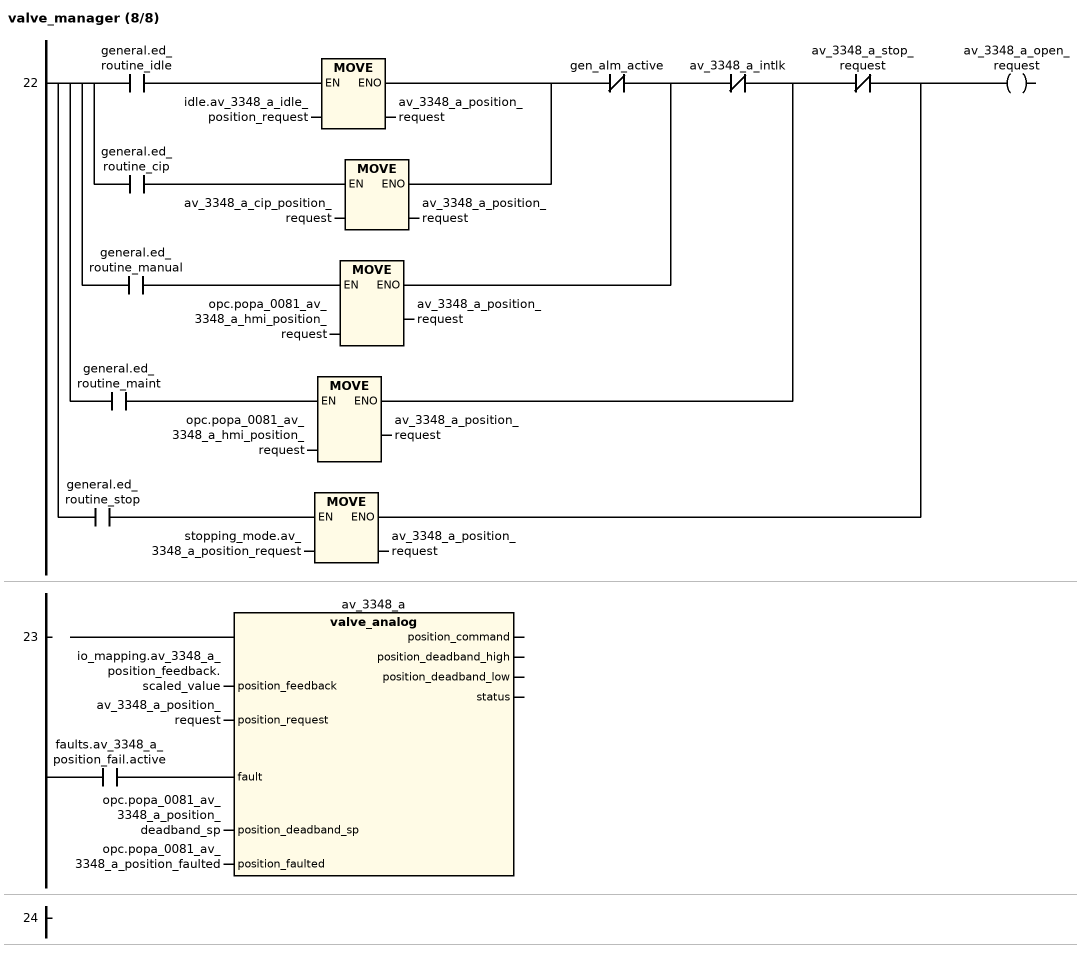
// NETWORK 22
_w11 := general.ed_routine_idle;
IF _w11 THEN av_3348_a_position_request := idle.av_3348_a_idle_position_request; END_IF
_w12 := general.ed_routine_cip;
IF _w12 THEN av_3348_a_position_request := av_3348_a_cip_position_request; END_IF
_w13 := general.ed_routine_manual;
IF _w13 THEN av_3348_a_position_request := opc.popa_0081_av_3348_a_hmi_position_request; END_IF
_w14 := general.ed_routine_maint;
IF _w14 THEN av_3348_a_position_request := opc.popa_0081_av_3348_a_hmi_position_request; END_IF
_w15 := general.ed_routine_stop;
IF _w15 THEN av_3348_a_position_request := stopping_mode.av_3348_a_position_request; END_IF
av_3348_a_open_request := (((_w11 OR _w12) AND NOT gen_alm_active OR _w13) AND NOT av_3348_a_intlk OR _w14) AND NOT av_3348_a_stop_request OR _w15;

// NETWORK 23
av_3348_a(
    position_feedback := io_mapping.av_3348_a_position_feedback.scaled_value,
    position_request := av_3348_a_position_request,
    fault := faults.av_3348_a_position_fail.active,
    position_deadband_sp := opc.popa_0081_av_3348_a_position_deadband_sp,
    position_faulted := opc.popa_0081_av_3348_a_position_faulted); // valve_analog

// NETWORK 24

END_PROGRAM

// ---- POUs/example_loop_control.TcPOU
PROGRAM example_loop_control
VAR
	//Example run request for a starter motor.  This would be triggered by control loop logic
	u_3160_b_run_request : BOOL;
	
	//Example run request for a vfd motor.  This would be triggered by control loop logic
	u_3112_b_run_request : BOOL;
	//Example Speed Request for a vfd motor.  This would be set by control loop logic, normally a PID
	u_3112_b_speed_request : REAL;
	
	//Example position request for an analog valve.  This would be set by control loop logic, normally a PID
	av_3148_b_position_request : REAL;
	
	//Example open request for a digital valve.  This would be triggered by control loop logic
	nv_3372_b_open_request : BOOL;
END_VAR

// NETWORK 1

END_PROGRAM

// ---- POUs/opc_control.TcPOU
PROGRAM opc_control
VAR PERSISTENT
	//Get Current Task Function, used in first scan bit logic
	get_current_task_index : GETCURTASKINDEX;
	//first scan bit, only true for one scan when system is activated/powered up
	first_scan_bit : BOOL;
	//OPC UA Server function, used for resetting server on activation
	opc_ua_server_command : FB_OpcUAServer;
	//Tells the OPC UA server what we want it to do, in this case restart
	server_command_option : E_OPCUAServerOption :=eOPCUAServerOption_Restart;
	//OPC UA Server command timeout
	timeout_setpoint: TIME :=T#30S;
	
	//Finds the AMS Net ID of the OPC UA server, in this case the local PLC
	get_local_ams_net_id: fb_getlocalamsnetid;
	//Toggle to request the ams net id
	amsnetid_request_started: BOOL;
	//Local AMS Net id of the PLC
	ams_net_id : T_AmsNetID;
	
END_VAR

//This logic is only needed for Windows CE based systems, like the CX-9020.  They do not restart the OPC server on activation, which means you need to manually restart the OPC server any time you make OPC changes.
//This logic automatically restarts the OPC server every time you activate the configuration, so you don't havd to do it manually.
//This is not required for larger, non-CE based systems like the CX-6030

//Instantiate the GetCurTaskIndex Function block, used in first scan bit
get_current_task_index();
//Instantiate the OPCUA Server Function Block
opc_ua_server_command();
//Set the OPC UA Server Command
opc_ua_server_command.eOpcUAServerOption:=server_command_option;
//Instantiate the Get Local AMS Net ID Function Block
get_local_ams_net_id();

//Get the local AMS Net ID.  This constantly toggles the request_started bit, to pull the Net ID continuously.
IF(amsnetid_request_started = FALSE) THEN
	get_local_ams_net_id(bexecute := TRUE, ttimeout := T#2S);
	amsnetid_request_started := TRUE;
ELSE
	IF(NOT get_local_ams_net_id.bBusy) THEN
		ams_net_id := get_local_ams_net_id.AddrString;
		get_local_ams_net_id.bExecute :=FALSE;
		amsnetid_request_started :=FALSE;
		END_IF
END_IF

//This sets the first scan bit true on first scan
IF _TaskInfo[get_current_task_index.index].FirstCycle THEN
	first_scan_bit:=TRUE;
END_IF

//Set the netid, execute, and timeout of the server command to the appropriate points, this is what actually resets the server on first scan
opc_ua_server_command.sNetId:=ams_net_id;
opc_ua_server_command.bExecute:=first_scan_bit;
opc_ua_server_command.tTimeout:=timeout_setpoint;

//Set the first scan bit back to false after the first scan
first_scan_bit:=FALSE;

END_PROGRAM

// ---- POUs/opc_mapping.TcPOU
PROGRAM opc_mapping
VAR
END_VAR

//This program maps values from the local variable to the OPC readable tag.
//Setpoints should NOT be mapped here.  The OPC tag should be used directly where needed
opc.popa_0081_av_3148_a_position_fail_active :=faults.av_3148_a_position_fail.active;
opc.popa_0081_u_3112_a_fail_to_start_active:=faults.u_3112_a_fail_to_start.active;
opc.popa_0081_u_3112_a_fail_to_stop_active:=faults.u_3112_a_fail_to_stop.active;
opc.popa_0081_u_3160_a_fail_to_start_active:=faults.u_3160_a_fail_to_start.active;
opc.popa_0081_u_3160_a_fail_to_stop_active:=faults.u_3112_a_fail_to_stop.active;
opc.popa_0081_cpt_3144_a_low_low_active:=faults.cpt_3144_a_low_low.active;
opc.popa_0081_cpt_3144_a_low_active:=faults.cpt_3144_a_low.active;
opc.popa_0081_cpt_3144_a_high_active:=faults.cpt_3144_a_high.active;
opc.popa_0081_cpt_3144_a_high_high_active:=faults.cpt_3144_a_high_high.active;

opc.popa_0081_ed_routine_critical_stop := general.ed_critical_stop;
opc.popa_0081_ed_routine_stop := general.ed_routine_stop;
opc.popa_0081_ed_routine_idle := general.ed_routine_idle;
opc.popa_0081_ed_routine_maint := general.ed_routine_maint;
opc.popa_0081_ed_routine_cip := general.ed_routine_cip;

opc.popa_0081_system_date_time_year:=general.system_date_time.year;
opc.popa_0081_system_date_time_month:=general.system_date_time.month;
opc.popa_0081_system_date_time_day:=general.system_date_time.day;
opc.popa_0081_system_date_time_hour:=general.system_date_time.hour;
opc.popa_0081_system_date_time_minute:=general.system_date_time.minute;
opc.popa_0081_system_date_time_second:=general.system_date_time.second;

//---Field Instrumentation---------------------------------------------------------------------------------------------------------------------------
opc.popa_0081_cpt_3144_a_scaled_value:=io_mapping.cpt_3144_a.scaled_value;

opc.popa_0081_ft_3122_a_scaled_value:=io_mapping.ft_3122_a.scaled_value;
opc.popa_0081_ft_3222_a_scaled_value:=io_mapping.ft_3222_a.scaled_value;
opc.popa_0081_ft_3322_a_scaled_value:=io_mapping.ft_3322_a.scaled_value;

opc.popa_0081_lt_3102_a_scaled_value:=io_mapping.lt_3102_a.scaled_value;
opc.popa_0081_lt_3202_a_scaled_value:=io_mapping.lt_3202_a.scaled_value;
opc.popa_0081_lt_3302_a_scaled_value:=io_mapping.lt_3302_a.scaled_value;
opc.popa_0081_lt_3153_a_scaled_value:=io_mapping.lt_3153_a.scaled_value;
opc.popa_0081_lt_3253_a_scaled_value:=io_mapping.lt_3253_a.scaled_value;
opc.popa_0081_lt_3353_a_scaled_value:=io_mapping.lt_3353_a.scaled_value;
opc.popa_0091_lt_3402_a_scaled_value:=io_mapping.lt_3402_a.scaled_value;

opc.popa_0081_pt_3119_a_scaled_value:=io_mapping.pt_3119_a.scaled_value;
opc.popa_0081_pt_3219_a_scaled_value:=io_mapping.pt_3219_a.scaled_value;
opc.popa_0081_pt_3319_a_scaled_value:=io_mapping.pt_3319_a.scaled_value;
opc.popa_0081_pt_3141_a_scaled_value:=io_mapping.pt_3141_a.scaled_value;
opc.popa_0081_pt_3241_a_scaled_value:=io_mapping.pt_3241_a.scaled_value;
opc.popa_0081_pt_3341_a_scaled_value:=io_mapping.pt_3341_a.scaled_value;
opc.popa_0091_pt_3428_a_scaled_value:=io_mapping.pt_3428_a.scaled_value;
opc.popa_0091_pt_3414_a_scaled_value:=io_mapping.pt_3414_a.scaled_value;

opc.popa_0081_tt_3118_a_scaled_value:=io_mapping.tt_3118_a.scaled_value;
opc.popa_0081_tt_3218_a_scaled_value:=io_mapping.tt_3218_a.scaled_value;
opc.popa_0081_tt_3318_a_scaled_value:=io_mapping.tt_3318_a.scaled_value;
opc.popa_0081_tt_3140_a_scaled_value:=io_mapping.tt_3140_a.scaled_value;
opc.popa_0081_tt_3240_a_scaled_value:=io_mapping.tt_3240_a.scaled_value;
opc.popa_0081_tt_3340_a_scaled_value:=io_mapping.tt_3340_a.scaled_value;
opc.popa_0091_tt_3432_a_scaled_value:=io_mapping.tt_3432_a.scaled_value;

//---Pumps---------------------------------------------------------------------------------------------------------------
opc.popa_0081_u_3112_a_speed_command_scaled_value:=output_mapping.u_3112_a_speed_command.scaled_value;
opc.popa_0081_u_3112_a_speed_feedback_scaled_value:=io_mapping.u_3112_a_speed_feedback.scaled_value;
opc.popa_0081_u_3112_a_run_request:=pump_manager.u_3112_a.run_request;
opc.popa_0081_u_3112_a_speed_request:=pump_manager.u_3112_a.speed_request;
opc.popa_0081_u_3112_a_runtime_today:=pump_manager.u_3112_a.runtime_today;
opc.popa_0081_u_3112_a_runtime_total:=pump_manager.u_3112_a.runtime_total;
opc.popa_0081_u_3112_a_runtime_maint:=pump_manager.u_3112_a.runtime_maint;
opc.popa_0081_u_3112_a_status:=pump_manager.u_3112_a.status;

opc.popa_0081_u_3212_a_speed_command_scaled_value:=output_mapping.u_3212_a_speed_command.scaled_value;
opc.popa_0081_u_3212_a_speed_feedback_scaled_value:=io_mapping.u_3212_a_speed_feedback.scaled_value;
opc.popa_0081_u_3212_a_run_request:=pump_manager.u_3212_a.run_request;
opc.popa_0081_u_3212_a_speed_request:=pump_manager.u_3212_a.speed_request;
opc.popa_0081_u_3212_a_runtime_today:=pump_manager.u_3212_a.runtime_today;
opc.popa_0081_u_3212_a_runtime_total:=pump_manager.u_3212_a.runtime_total;
opc.popa_0081_u_3212_a_runtime_maint:=pump_manager.u_3212_a.runtime_maint;
opc.popa_0081_u_3212_a_status:=pump_manager.u_3212_a.status;

opc.popa_0081_u_3312_a_speed_command_scaled_value:=output_mapping.u_3312_a_speed_command.scaled_value;
opc.popa_0081_u_3312_a_speed_feedback_scaled_value:=io_mapping.u_3312_a_speed_feedback.scaled_value;
opc.popa_0081_u_3312_a_run_request:=pump_manager.u_3312_a.run_request;
opc.popa_0081_u_3312_a_speed_request:=pump_manager.u_3312_a.speed_request;
opc.popa_0081_u_3312_a_runtime_today:=pump_manager.u_3312_a.runtime_today;
opc.popa_0081_u_3312_a_runtime_total:=pump_manager.u_3312_a.runtime_total;
opc.popa_0081_u_3312_a_runtime_maint:=pump_manager.u_3312_a.runtime_maint;
opc.popa_0081_u_3312_a_status:=pump_manager.u_3312_a.status;

opc.popa_0081_u_3160_a_speed_command_scaled_value:=output_mapping.u_3160_a_speed_command.scaled_value;
opc.popa_0081_u_3160_a_speed_feedback_scaled_value:=io_mapping.u_3160_a_speed_feedback.scaled_value;
opc.popa_0081_u_3160_a_run_request:=pump_manager.u_3160_a.run_request;
opc.popa_0081_u_3160_a_speed_request:=pump_manager.u_3160_a.speed_request;
opc.popa_0081_u_3160_a_runtime_today:=pump_manager.u_3160_a.runtime_today;
opc.popa_0081_u_3160_a_runtime_total:=pump_manager.u_3160_a.runtime_total;
opc.popa_0081_u_3160_a_runtime_maint:=pump_manager.u_3160_a.runtime_maint;
opc.popa_0081_u_3160_a_status:=pump_manager.u_3160_a.status;

opc.popa_0081_u_3260_a_speed_command_scaled_value:=output_mapping.u_3260_a_speed_command.scaled_value;
opc.popa_0081_u_3260_a_speed_feedback_scaled_value:=io_mapping.u_3260_a_speed_feedback.scaled_value;
opc.popa_0081_u_3260_a_run_request:=pump_manager.u_3260_a.run_request;
opc.popa_0081_u_3260_a_speed_request:=pump_manager.u_3260_a.speed_request;
opc.popa_0081_u_3260_a_runtime_today:=pump_manager.u_3260_a.runtime_today;
opc.popa_0081_u_3260_a_runtime_total:=pump_manager.u_3260_a.runtime_total;
opc.popa_0081_u_3260_a_runtime_maint:=pump_manager.u_3260_a.runtime_maint;
opc.popa_0081_u_3260_a_status:=pump_manager.u_3260_a.status;

opc.popa_0081_u_3360_a_speed_command_scaled_value:=output_mapping.u_3360_a_speed_command.scaled_value;
opc.popa_0081_u_3360_a_speed_feedback_scaled_value:=io_mapping.u_3360_a_speed_feedback.scaled_value;
opc.popa_0081_u_3360_a_run_request:=pump_manager.u_3360_a.run_request;
opc.popa_0081_u_3360_a_speed_request:=pump_manager.u_3360_a.speed_request;
opc.popa_0081_u_3360_a_runtime_today:=pump_manager.u_3360_a.runtime_today;
opc.popa_0081_u_3360_a_runtime_total:=pump_manager.u_3360_a.runtime_total;
opc.popa_0081_u_3360_a_runtime_maint:=pump_manager.u_3360_a.runtime_maint;
opc.popa_0081_u_3360_a_status:=pump_manager.u_3360_a.status;

opc.popa_0081_u_3370_a_speed_command_scaled_value:=output_mapping.u_3370_a_speed_command.scaled_value;
opc.popa_0081_u_3370_a_speed_feedback_scaled_value:=io_mapping.u_3370_a_speed_feedback.scaled_value;
opc.popa_0081_u_3370_a_run_request:=pump_manager.u_3370_a.run_request;
opc.popa_0081_u_3370_a_speed_request:=pump_manager.u_3370_a.speed_request;
opc.popa_0081_u_3370_a_runtime_today:=pump_manager.u_3370_a.runtime_today;
opc.popa_0081_u_3370_a_runtime_total:=pump_manager.u_3370_a.runtime_total;
opc.popa_0081_u_3370_a_runtime_maint:=pump_manager.u_3370_a.runtime_maint;
opc.popa_0081_u_3370_a_status:=pump_manager.u_3370_a.status;

opc.popa_0091_u_3405_a_speed_command_scaled_value:=output_mapping.u_3405_a_speed_command.scaled_value;
opc.popa_0091_u_3405_a_speed_feedback_scaled_value:=io_mapping.u_3405_a_speed_feedback.scaled_value;
opc.popa_0091_u_3405_a_run_request:=pump_manager.u_3405_a.run_request;
opc.popa_0091_u_3405_a_speed_request:=pump_manager.u_3405_a.speed_request;
opc.popa_0091_u_3405_a_runtime_today:=pump_manager.u_3405_a.runtime_today;
opc.popa_0091_u_3405_a_runtime_total:=pump_manager.u_3405_a.runtime_total;
opc.popa_0091_u_3405_a_runtime_maint:=pump_manager.u_3405_a.runtime_maint;
opc.popa_0091_u_3405_a_status:=pump_manager.u_3405_a.status;



//---Valves------------------------------------------------------------------------------------------------------------------

opc.popa_0081_av_3148_a_position_feedback_scaled_value:=io_mapping.av_3148_a_position_feedback.scaled_value;
opc.popa_0081_av_3148_a_position_command_scaled_value:=output_mapping.av_3148_a_position_command.scaled_value;
opc.popa_0081_av_3148_a_position_feedback:=valve_manager.av_3148_a.position_feedback;
opc.popa_0081_av_3148_a_position_request:=valve_manager.av_3148_a.position_request;
opc.popa_0081_av_3148_a_status:=valve_manager.av_3148_a.status;

opc.popa_0081_av_3248_a_position_feedback_scaled_value:=io_mapping.av_3248_a_position_feedback.scaled_value;
opc.popa_0081_av_3248_a_position_command_scaled_value:=output_mapping.av_3248_a_position_command.scaled_value;
opc.popa_0081_av_3248_a_position_feedback:=valve_manager.av_3248_a.position_feedback;
opc.popa_0081_av_3248_a_position_request:=valve_manager.av_3248_a.position_request;
opc.popa_0081_av_3248_a_status:=valve_manager.av_3248_a.status;

opc.popa_0081_av_3348_a_position_feedback_scaled_value:=io_mapping.av_3348_a_position_feedback.scaled_value;
opc.popa_0081_av_3348_a_position_command_scaled_value:=output_mapping.av_3348_a_position_command.scaled_value;
opc.popa_0081_av_3348_a_position_feedback:=valve_manager.av_3348_a.position_feedback;
opc.popa_0081_av_3348_a_position_request:=valve_manager.av_3348_a.position_request;
opc.popa_0081_av_3348_a_status:=valve_manager.av_3348_a.status;
(*
opc.popa_0081_u_3160_a_run_request:=motor_starter_control.u_3160_a.run_request;
opc.popa_0081_u_3160_a_runtime_today:=motor_starter_control.u_3160_a.runtime_today;
opc.popa_0081_u_3160_a_runtime_total:=motor_starter_control.u_3160_a.runtime_total;
opc.popa_0081_u_3160_a_runtime_maint:=motor_starter_control.u_3160_a.runtime_maint;
opc.popa_0081_u_3160_a_status:=motor_starter_control.u_3160_a.status;
*)


opc.popa_0081_nv_3110_a_open_request:=valve_manager.nv_3110_a.open_request;
opc.popa_0081_nv_3110_a_status:=valve_manager.nv_3110_a.status;
opc.popa_0081_nv_3110_a_fail_to_open_active :=faults.nv_3110_a_fail_to_open.active;
opc.popa_0081_nv_3110_a_fail_to_close_active :=faults.nv_3110_a_fail_to_close.active;

opc.popa_0081_nv_3210_a_open_request:=valve_manager.nv_3210_a.open_request;
opc.popa_0081_nv_3210_a_status:=valve_manager.nv_3210_a.status;
opc.popa_0081_nv_3210_a_fail_to_open_active :=faults.nv_3210_a_fail_to_open.active;
opc.popa_0081_nv_3210_a_fail_to_close_active :=faults.nv_3210_a_fail_to_close.active;

opc.popa_0081_nv_3310_a_open_request:=valve_manager.nv_3310_a.open_request;
opc.popa_0081_nv_3310_a_status:=valve_manager.nv_3310_a.status;
opc.popa_0081_nv_3310_a_fail_to_open_active :=faults.nv_3310_a_fail_to_open.active;
opc.popa_0081_nv_3310_a_fail_to_close_active :=faults.nv_3310_a_fail_to_close.active;

opc.popa_0081_nv_3135_a_open_request:=valve_manager.nv_3135_a.open_request;
opc.popa_0081_nv_3135_a_status:=valve_manager.nv_3135_a.status;
opc.popa_0081_nv_3135_a_fail_to_open_active :=faults.nv_3135_a_fail_to_open.active;
opc.popa_0081_nv_3135_a_fail_to_close_active :=faults.nv_3135_a_fail_to_close.active;

opc.popa_0081_nv_3235_a_open_request:=valve_manager.nv_3235_a.open_request;
opc.popa_0081_nv_3235_a_status:=valve_manager.nv_3235_a.status;
opc.popa_0081_nv_3235_a_fail_to_open_active :=faults.nv_3235_a_fail_to_open.active;
opc.popa_0081_nv_3235_a_fail_to_close_active :=faults.nv_3235_a_fail_to_close.active;

opc.popa_0081_nv_3335_a_open_request:=valve_manager.nv_3335_a.open_request;
opc.popa_0081_nv_3335_a_status:=valve_manager.nv_3335_a.status;
opc.popa_0081_nv_3335_a_fail_to_open_active :=faults.nv_3335_a_fail_to_open.active;
opc.popa_0081_nv_3335_a_fail_to_close_active :=faults.nv_3335_a_fail_to_close.active;

opc.popa_0081_nv_3372_a_open_request:=valve_manager.nv_3372_a.open_request;
opc.popa_0081_nv_3372_a_status:=valve_manager.nv_3372_a.status;
opc.popa_0081_nv_3372_a_fail_to_open_active :=faults.nv_3372_a_fail_to_open.active;
opc.popa_0081_nv_3372_a_fail_to_close_active :=faults.nv_3372_a_fail_to_close.active;

//opc.popa_0081_nv_3162_a_hmi_open_request:=valve_manager.nv_3162_a.open_request;
opc.popa_0081_nv_3162_a_open_request:=valve_manager.nv_3162_a.open_request;
opc.popa_0081_nv_3162_a_status:=valve_manager.nv_3162_a.status;
opc.popa_0081_nv_3162_a_fail_to_open_active :=faults.nv_3162_a_fail_to_open.active;
opc.popa_0081_nv_3162_a_fail_to_close_active :=faults.nv_3162_a_fail_to_close.active;

END_PROGRAM

// ---- POUs/output_mapping.TcPOU
PROGRAM output_mapping
VAR PERSISTENT
	//Motor vfd speed command function block
	u_3112_a_speed_command : analog_scaling;
	u_3212_a_speed_command : analog_scaling;
	u_3312_a_speed_command : analog_scaling;
	u_3160_a_speed_command : analog_scaling;
	u_3260_a_speed_command : analog_scaling;
	u_3360_a_speed_command : analog_scaling;
	u_3370_a_speed_command : analog_scaling;
	u_3405_a_speed_command : analog_scaling;
	
	//Analog valve position command
	av_3148_a_position_command : analog_scaling;
	av_3248_a_position_command : analog_scaling;
	av_3348_a_position_command : analog_scaling;
	nv_3110_a_position_command : analog_scaling;
	nv_3210_a_position_command : analog_scaling;
	nv_3310_a_position_command : analog_scaling;
	//Motor vfd speed command scaled output, mappped to a physical output
	{attribute 'TcLinkTo' := 'TIID^Device 1 (EtherCAT)^Term 1 (EK1200)^Term 4 (EL4124)^AO Output Channel 1^Analog output'}
	u_3112_a_speed_command_io AT %Q* : INT;
	{attribute 'TcLinkTo' := 'TIID^Device 1 (EtherCAT)^Term 1 (EK1200)^Term 4 (EL4124)^AO Output Channel 2^Analog output'}
	u_3212_a_speed_command_io AT %Q* : INT;
	{attribute 'TcLinkTo' := 'TIID^Device 1 (EtherCAT)^Term 1 (EK1200)^Term 4 (EL4124)^AO Output Channel 3^Analog output'}
	u_3312_a_speed_command_io AT %Q* : INT;
	{attribute 'TcLinkTo' := 'TIID^Device 1 (EtherCAT)^Term 1 (EK1200)^Term 4 (EL4124)^AO Output Channel 4^Analog output'}
	u_3160_a_speed_command_io AT %Q* : INT;
	{attribute 'TcLinkTo' := 'TIID^Device 1 (EtherCAT)^Term 1 (EK1200)^Term 5 (EL4124)^AO Output Channel 1^Analog output'}
	u_3260_a_speed_command_io AT %Q* : INT;
	{attribute 'TcLinkTo' := 'TIID^Device 1 (EtherCAT)^Term 1 (EK1200)^Term 5 (EL4124)^AO Output Channel 2^Analog output'}
	u_3360_a_speed_command_io AT %Q* : INT;
	{attribute 'TcLinkTo' := 'TIID^Device 1 (EtherCAT)^Term 1 (EK1200)^Term 5 (EL4124)^AO Output Channel 3^Analog output'}
	u_3370_a_speed_command_io AT %Q* : INT;
	{attribute 'TcLinkTo' := 'TIID^Device 1 (EtherCAT)^Term 40 (EK1100)^Term 42 (EL4124)^AO Output Channel 1^Analog output'}
	u_3405_a_speed_command_io AT %Q* : INT;
	
	//Motor vfd run command, mapped to a physical output
	{attribute 'TcLinkTo' :=  'TIID^Device 1 (EtherCAT)^Term 1 (EK1200)^Term 7 (EL1859)^Channel 9^Output'}
	u_3112_a_run_command_io AT %Q* : BOOL;
	{attribute 'TcLinkTo' :=  'TIID^Device 1 (EtherCAT)^Term 1 (EK1200)^Term 7 (EL1859)^Channel 11^Output'}
	u_3212_a_run_command_io AT %Q* : BOOL;
	{attribute 'TcLinkTo' :=  'TIID^Device 1 (EtherCAT)^Term 1 (EK1200)^Term 7 (EL1859)^Channel 13^Output'}
	u_3312_a_run_command_io AT %Q* : BOOL;
	{attribute 'TcLinkTo' :=  'TIID^Device 1 (EtherCAT)^Term 1 (EK1200)^Term 7 (EL1859)^Channel 15^Output'}	
	u_3160_a_run_command_io AT %Q* : BOOL;
	{attribute 'TcLinkTo' :=  'TIID^Device 1 (EtherCAT)^Term 1 (EK1200)^Term 8 (EL1859)^Channel 9^Output'}
	u_3260_a_run_command_io AT %Q* : BOOL;
	{attribute 'TcLinkTo' :=  'TIID^Device 1 (EtherCAT)^Term 1 (EK1200)^Term 8 (EL1859)^Channel 11^Output'}
	u_3360_a_run_command_io AT %Q* : BOOL;
	{attribute 'TcLinkTo' :=  'TIID^Device 1 (EtherCAT)^Term 1 (EK1200)^Term 8 (EL1859)^Channel 13^Output'}
	u_3370_a_run_command_io AT %Q* : BOOL;
	{attribute 'TcLinkTo' :=  'TIID^Device 1 (EtherCAT)^Term 40 (EK1100)^Term 43 (EL1859)^Channel 9^Output'}
	u_3405_a_run_command_io AT %Q* : BOOL;
	
	//Motor Fault Reset
	{attribute 'TcLinkTo' :=  'TIID^Device 1 (EtherCAT)^Term 1 (EK1200)^Term 7 (EL1859)^Channel 10^Output'}
	u_3112_a_fault_reset_io AT %Q* : BOOL;
	{attribute 'TcLinkTo' :=  'TIID^Device 1 (EtherCAT)^Term 1 (EK1200)^Term 7 (EL1859)^Channel 12^Output'}
	u_3212_a_fault_reset_io AT %Q* : BOOL;
	{attribute 'TcLinkTo' :=  'TIID^Device 1 (EtherCAT)^Term 1 (EK1200)^Term 7 (EL1859)^Channel 14^Output'}
	u_3312_a_fault_reset_io AT %Q* : BOOL;
	{attribute 'TcLinkTo' :=  'TIID^Device 1 (EtherCAT)^Term 1 (EK1200)^Term 7 (EL1859)^Channel 16^Output'}
	u_3160_a_fault_reset_io AT %Q* : BOOL;
	{attribute 'TcLinkTo' :=  'TIID^Device 1 (EtherCAT)^Term 1 (EK1200)^Term 8 (EL1859)^Channel 10^Output'}
	u_3260_a_fault_reset_io AT %Q* : BOOL;
	{attribute 'TcLinkTo' :=  'TIID^Device 1 (EtherCAT)^Term 1 (EK1200)^Term 8 (EL1859)^Channel 12^Output'}
	u_3360_a_fault_reset_io AT %Q* : BOOL;
	{attribute 'TcLinkTo' :=  'TIID^Device 1 (EtherCAT)^Term 1 (EK1200)^Term 8 (EL1859)^Channel 14^Output'}
	u_3370_a_fault_reset_io AT %Q* : BOOL;
	{attribute 'TcLinkTo' :=  'TIID^Device 1 (EtherCAT)^Term 40 (EK1100)^Term 43 (EL1859)^Channel 10^Output'}
	u_3405_a_fault_reset_io AT %Q* : BOOL;
	
		
	//Analog valve position command output valve
	{attribute 'TcLinkTo' := 'TIID^Device 1 (EtherCAT)^Term 20 (EK1100-0018)^Term 26 (EL4124)^AO Output Channel 1^Analog output'}
	av_3148_a_position_command_io AT %Q* : INT;
	{attribute 'TcLinkTo' := 'TIID^Device 1 (EtherCAT)^Term 20 (EK1100-0018)^Term 26 (EL4124)^AO Output Channel 2^Analog output'}
	av_3248_a_position_command_io AT %Q* : INT;
	{attribute 'TcLinkTo' := 'TIID^Device 1 (EtherCAT)^Term 20 (EK1100-0018)^Term 26 (EL4124)^AO Output Channel 3^Analog output'}
	av_3348_a_position_command_io AT %Q* : INT;
	
		//Digital valve open command
	{attribute 'TcLinkTo' := 'TIID^Device 1 (EtherCAT)^Term 31 (EK1914)^Term 32 (EL1859)^Channel 11^Output'}
	nv_3110_a_open_command_io AT %Q* : BOOL;
	{attribute 'TcLinkTo' := 'TIID^Device 1 (EtherCAT)^Term 31 (EK1914)^Term 32 (EL1859)^Channel 10^Output'}
	nv_3210_a_open_command_io AT %Q* : BOOL;
	{attribute 'TcLinkTo' := 'TIID^Device 1 (EtherCAT)^Term 31 (EK1914)^Term 32 (EL1859)^Channel 13^Output'}
	nv_3310_a_open_command_io AT %Q* : BOOL;
	{attribute 'TcLinkTo' := 'TIID^Device 1 (EtherCAT)^Term 31 (EK1914)^Term 32 (EL1859)^Channel 12^Output'}
	nv_3135_a_open_command_io AT %Q* : BOOL;
	{attribute 'TcLinkTo' := 'TIID^Device 1 (EtherCAT)^Term 31 (EK1914)^Term 32 (EL1859)^Channel 14^Output'}
	nv_3235_a_open_command_io AT %Q* : BOOL;
	{attribute 'TcLinkTo' := 'TIID^Device 1 (EtherCAT)^Term 31 (EK1914)^Term 32 (EL1859)^Channel 15^Output'}
	nv_3335_a_open_command_io AT %Q* : BOOL;
	{attribute 'TcLinkTo' := 'TIID^Device 1 (EtherCAT)^Term 31 (EK1914)^Term 32 (EL1859)^Channel 16^Output'}
	nv_3372_a_open_command_io AT %Q* : BOOL;
	{attribute 'TcLinkTo' := 'TIID^Device 1 (EtherCAT)^Term 31 (EK1914)^Term 32 (EL1859)^Channel 9^Output'}
	nv_3162_a_open_command_io AT %Q* : BOOL;
	
	safety_reset AT %Q* : BOOL;
END_VAR

//Map the motor run command to the command output
u_3112_a_run_command_io:=pump_manager.u_3112_a.run_command;
u_3212_a_run_command_io:=pump_manager.u_3212_a.run_command;
u_3312_a_run_command_io:=pump_manager.u_3312_a.run_command;
u_3160_a_run_command_io:=pump_manager.u_3160_a.run_command;
u_3260_a_run_command_io:=pump_manager.u_3260_a.run_command;
u_3360_a_run_command_io:=pump_manager.u_3360_a.run_command;
u_3370_a_run_command_io:=pump_manager.u_3370_a.run_command;
u_3405_a_run_command_io:=pump_manager.u_3405_a.run_command;

//Instantiate u_3112 Speed command analog output function block
u_3112_a_speed_command();
//Map values from the OPC GVL so that they can be written to from outside POU(IE from HMI)
u_3112_a_speed_command.eu_max:=32767;
u_3112_a_speed_command.eu_min:=0;
u_3112_a_speed_command.filter_factor:=opc.popa_0081_u_3112_a_speed_command_filter_factor;
u_3112_a_speed_command.raw_max:=60;
u_3112_a_speed_command.raw_min:=0;

//Map output from motor control pou to scaling block
u_3112_a_speed_command.raw_input := pump_manager.u_3112_a.speed_command;

//Map the analog scaling function block raw input to the physical raw output variable
u_3112_a_speed_command_io := REAL_TO_INT(u_3112_a_speed_command.scaled_value);

//Instantiate Example analog output function block
u_3212_a_speed_command();
//Map values from the OPC GVL so that they can be written to from outside POU(IE from HMI)
u_3212_a_speed_command.eu_max:=32767;
u_3212_a_speed_command.eu_min:=0;
u_3212_a_speed_command.filter_factor:=opc.popa_0081_u_3212_a_speed_command_filter_factor;
u_3212_a_speed_command.raw_max:=60;
u_3212_a_speed_command.raw_min:=0;

//Map output from motor control pou to scaling block
u_3212_a_speed_command.raw_input := pump_manager.u_3212_a.speed_command;

//Map the analog scaling function block raw input to the physical raw output variable
u_3212_a_speed_command_io := REAL_TO_INT(u_3212_a_speed_command.scaled_value);


//Instantiate Example analog output function block
u_3312_a_speed_command();
//Map values from the OPC GVL so that they can be written to from outside POU(IE from HMI)
u_3312_a_speed_command.eu_max:=32767;
u_3312_a_speed_command.eu_min:=0;
u_3312_a_speed_command.filter_factor:=opc.popa_0081_u_3312_a_speed_command_filter_factor;
u_3312_a_speed_command.raw_max:=60;
u_3312_a_speed_command.raw_min:=0;

//Map output from motor control pou to scaling block
u_3312_a_speed_command.raw_input := pump_manager.u_3312_a.speed_command;

//Map the analog scaling function block raw input to the physical raw output variable
u_3312_a_speed_command_io := REAL_TO_INT(u_3312_a_speed_command.scaled_value);


//Instantiate Example analog output function block
u_3160_a_speed_command();
//Map values from the OPC GVL so that they can be written to from outside POU(IE from HMI)
u_3160_a_speed_command.eu_max:=32767;
u_3160_a_speed_command.eu_min:=0;
u_3160_a_speed_command.filter_factor:=opc.popa_0081_u_3160_a_speed_command_filter_factor;
u_3160_a_speed_command.raw_max:=60;
u_3160_a_speed_command.raw_min:=0;

//Map output from motor control pou to scaling block
u_3160_a_speed_command.raw_input := pump_manager.u_3160_a.speed_command;

//Map the analog scaling function block raw input to the physical raw output variable
u_3160_a_speed_command_io := REAL_TO_INT(u_3160_a_speed_command.scaled_value);

//Instantiate Example analog output function block
u_3260_a_speed_command();
//Map values from the OPC GVL so that they can be written to from outside POU(IE from HMI)
u_3260_a_speed_command.eu_max:=32767;
u_3260_a_speed_command.eu_min:=0;
u_3260_a_speed_command.filter_factor:=opc.popa_0081_u_3260_a_speed_command_filter_factor;
u_3260_a_speed_command.raw_max:=60;
u_3260_a_speed_command.raw_min:=0;

//Map output from motor control pou to scaling block
u_3260_a_speed_command.raw_input := pump_manager.u_3260_a.speed_command;

//Map the analog scaling function block raw input to the physical raw output variable
u_3260_a_speed_command_io := REAL_TO_INT(u_3260_a_speed_command.scaled_value);

//Instantiate Example analog output function block
u_3360_a_speed_command();
//Map values from the OPC GVL so that they can be written to from outside POU(IE from HMI)
u_3360_a_speed_command.eu_max:=32767;
u_3360_a_speed_command.eu_min:=0;
u_3360_a_speed_command.filter_factor:=opc.popa_0081_u_3360_a_speed_command_filter_factor;
u_3360_a_speed_command.raw_max:=60;
u_3360_a_speed_command.raw_min:=0;

//Map output from motor control pou to scaling block
u_3360_a_speed_command.raw_input := pump_manager.u_3360_a.speed_command;

//Map the analog scaling function block raw input to the physical raw output variable
u_3360_a_speed_command_io := REAL_TO_INT(u_3360_a_speed_command.scaled_value);


//Instantiate Example analog output function block
u_3370_a_speed_command();
//Map values from the OPC GVL so that they can be written to from outside POU(IE from HMI)
u_3370_a_speed_command.eu_max:=32767;
u_3370_a_speed_command.eu_min:=0;
u_3370_a_speed_command.filter_factor:=opc.popa_0081_u_3370_a_speed_command_filter_factor;
u_3370_a_speed_command.raw_max:=60;
u_3370_a_speed_command.raw_min:=0;

//Map output from motor control pou to scaling block
u_3370_a_speed_command.raw_input := pump_manager.u_3370_a.speed_command;

//Map the analog scaling function block raw input to the physical raw output variable
u_3370_a_speed_command_io := REAL_TO_INT(u_3370_a_speed_command.scaled_value);

//Instantiate Example analog output function block
u_3405_a_speed_command();
//Map values from the OPC GVL so that they can be written to from outside POU(IE from HMI)
u_3405_a_speed_command.eu_max:=32767;
u_3405_a_speed_command.eu_min:=0;
u_3405_a_speed_command.filter_factor:=opc.popa_0091_u_3405_a_speed_command_filter_factor;
u_3405_a_speed_command.raw_max:=60;
u_3405_a_speed_command.raw_min:=0;

//Map output from motor control pou to scaling block
u_3405_a_speed_command.raw_input := pump_manager.u_3405_a.speed_command;

//Map the analog scaling function block raw input to the physical raw output variable
u_3405_a_speed_command_io := REAL_TO_INT(u_3405_a_speed_command.scaled_value);

//Instantiate av_3148 analog output function block
av_3148_a_position_command();
//Map values from the OPC GVL so that they can be written to from outside POU(IE from HMI)
av_3148_a_position_command.eu_max:=32767;
av_3148_a_position_command.eu_min:=0;
av_3148_a_position_command.filter_factor:=opc.popa_0081_av_3148_a_position_command_filter_factor;
av_3148_a_position_command.raw_max:=100;
av_3148_a_position_command.raw_min:=0;
//Map output from valve control pou to scaling block
av_3148_a_position_command.raw_input:=valve_manager.av_3148_a.Position_Command;
//Map the analog scaling function block raw input to the physical raw output variable
av_3148_a_position_command_io := REAL_TO_INT(av_3148_a_position_command.scaled_value);

//Instantiate av_3248 analog output function block
av_3248_a_position_command();
//Map values from the OPC GVL so that they can be written to from outside POU(IE from HMI)
av_3248_a_position_command.eu_max:=32767;
av_3248_a_position_command.eu_min:=0;
av_3248_a_position_command.filter_factor:=opc.popa_0081_av_3248_a_position_command_filter_factor;
av_3248_a_position_command.raw_max:=100;
av_3248_a_position_command.raw_min:=0;
//Map output from valve control pou to scaling block
av_3248_a_position_command.raw_input:=valve_manager.av_3248_a.Position_Command;
//Map the analog scaling function block raw input to the physical raw output variable
av_3248_a_position_command_io := REAL_TO_INT(av_3248_a_position_command.scaled_value);

//Instantiate av_3348 analog output function block
av_3348_a_position_command();
//Map values from the OPC GVL so that they can be written to from outside POU(IE from HMI)
av_3348_a_position_command.eu_max:=32767;
av_3348_a_position_command.eu_min:=0;
av_3348_a_position_command.filter_factor:=opc.popa_0081_av_3348_a_position_command_filter_factor;
av_3348_a_position_command.raw_max:=100;
av_3348_a_position_command.raw_min:=0;
//Map output from valve control pou to scaling block
av_3348_a_position_command.raw_input:=valve_manager.av_3348_a.Position_Command;
//Map the analog scaling function block raw input to the physical raw output variable
av_3348_a_position_command_io := REAL_TO_INT(av_3348_a_position_command.scaled_value);


//Map the digital valve open command to the command output
nv_3110_a_open_command_io:=valve_manager.nv_3110_a.open_command;
nv_3210_a_open_command_io:=valve_manager.nv_3210_a.open_command;
nv_3310_a_open_command_io:=valve_manager.nv_3310_a.open_command;
nv_3135_a_open_command_io:=valve_manager.nv_3135_a.open_command;
nv_3235_a_open_command_io:=valve_manager.nv_3235_a.open_command;
nv_3335_a_open_command_io:=valve_manager.nv_3335_a.open_command;
nv_3372_a_open_command_io:=valve_manager.nv_3372_a.open_command;
nv_3162_a_open_command_io:=valve_manager.nv_3162_a.open_command;

END_PROGRAM
